INTERFACE I_UnitTest EXTENDS __SYSTEM.IQueryInterface

METHOD Execute
END_METHOD

METHOD Initialise
VAR_INPUT
    MessageList : I_AssertionMessageList;
END_VAR
END_METHOD

PROPERTY TestHasFailed : BOOL
GET
END_GET
END_PROPERTY

PROPERTY TestHasFinished : BOOL
GET
END_GET
END_PROPERTY

PROPERTY TestName : T_MaxString
GET
END_GET
END_PROPERTY

END_INTERFACE

(* stored: Version 1.1.0.1, ProductVersion 3.1.4024.4
   Itf I_UnitTest: Id {137795db-abc7-4fa7-8556-f33fd38a5e22}
   Method Execute: Id {2fba04c3-dc29-45c8-9862-61e987437cae}
   Method Initialise: Id {c9388da0-0ae6-4f8c-8201-6c010a8515b8}
   Property TestHasFailed: Id {df9c8aa0-74e0-4748-8bd2-4a5fb0af13a5}
   Get Get: Id {1a2f703b-1650-4083-8e8e-2f36512fa429}
   Property TestHasFinished: Id {007eb33b-a04a-4cb1-8b1a-872bdd85f4d0}
   Get Get: Id {71a925c9-9c56-4b8d-b544-8cdd0a5a0cfa}
   Property TestName: Id {fca77da0-e028-4f06-adf6-809516ee7298}
   Get Get: Id {e1d0f475-1d5c-4058-8f2a-d47b2144376a} *)
